// TIA Portal V17 export
// export: Created 2023-12-22T15:08:00.0545629Z, ExportSetting WithDefaults, DisplayName Totally Integrated Automation Portal, DisplayVersion V17, DisplayName TIA Portal Openness, DisplayVersion V17, DisplayName TIA Portal Version Control Interface, DisplayVersion V17, DisplayName STEP 7 Professional, DisplayVersion V17, DisplayName STEP 7 Safety, DisplayVersion V17, DisplayName WinCC Advanced, DisplayVersion V17
FUNCTION_BLOCK "PS_One"   // FB11, LAD
{ S7_Optimized_Access := 'FALSE' }
VERSION : 0.1
// Mode - 0 - выкл, 1 - быстрый разгон, 2 - плавный разон, 3 - работа, 4 - притормозить для ввода нового насоса, 5 - замедлить плавно, 6 - замедлить быстро
// 
// Status - 0 выкл, 1 - быстро разгоняется, 10 - вышел на точку, 2 - плавно разгоняется, 20 - вышел на точку, 3 - в работе, 4 - притормаживается для выхода на общую точку, 40 - общая точка достигнута, 5 - замедлить для отключения, 50 - замедлено до нижней точки, 6 - вывести из работы через быстрый сброс оборотов, 60 - обороты сброшены и готов к отключению, 99 - насос в аварии/не готов к работе
// stored: AutoNumber false, IsIECCheckEnabled false, SetENOAutomatically false, UDAEnableTagReadback false
   VAR_INPUT
      in_PE : Real;   // Давление на всасывании
      P_FB_SP : Real;   // Текущая скорость / Уставка скорости для ЧП
      P_Alarm : Bool;   // Авария ЧП
      P_Warning : Bool;   // Предупреждение ЧП
   END_VAR
   VAR_OUTPUT
      P_CMD : Bool;   // Команда на ЧП
      P_SP : Real;   // Уставка на ЧП
      P_Step_Up : Real := 0.01;   // Шаг разгона для ЧП
      P_Step_Down : Real := 0.01;   // Шаг замедления для ЧП
   END_VAR
   VAR_IN_OUT
      P_Res : DInt;   // Наработка ЧП
   END_VAR
   VAR DB_SPECIFIC
      CMD : "CMD";   // Блок команд
      Min { S7_SetPoint := 'True'} : Bool;
      Max : Bool;
      PE_Warning : Bool;
      SP_A : Real;   // Уставка в авторежиме
      SP : Real;   // Фактическая уставка
      Mode : Int;   // Запрашиваемый режим работы
      Hand_Mode : Int := 3;   // Режим работы в ручном режиме
      Status : Int;   // Фактический режим работы
      Weight : Real;   // Коэфф. выбора насоса
      Start_per_H_SP : Int := 5;
      Start_per_H_Now : Int;
      Alarms : Word;
      Events : Word;
      pos : Array[0..15] of Bool;
   END_VAR
   VAR
      T_Delay { S7_SetPoint := 'True'} : "Time_M";   // Минимальная задержка между пусками
      T_PE_Delay { S7_SetPoint := 'True'} : "Time_M";
   END_VAR
   VAR_TEMP
      ev : Bool;
   END_VAR
   // T_Delay.SP_M := 10;
   // T_Delay.SP_S := 0;
   VAR_TEMP   // added for the SCL form of the ladder/FBD networks
      _w1 : Bool;
      _w2 : Bool;
      _w3 : Bool;
      _w4 : Bool;
      _w5 : Bool;
      _w6 : Bool;
      _w7 : Bool;
      _w8 : Bool;
      _w9 : Bool;
      _w10 : Bool;
      _w11 : Bool;
      _w12 : Bool;
      _w13 : Bool;
      _w14 : Bool;
      _w15 : Bool;
      _w16 : Bool;
      _w17 : Bool;
      _w18 : Bool;
      _w19 : Bool;
      _w20 : Bool;
   END_VAR
BEGIN

REGION Network 1: - - -
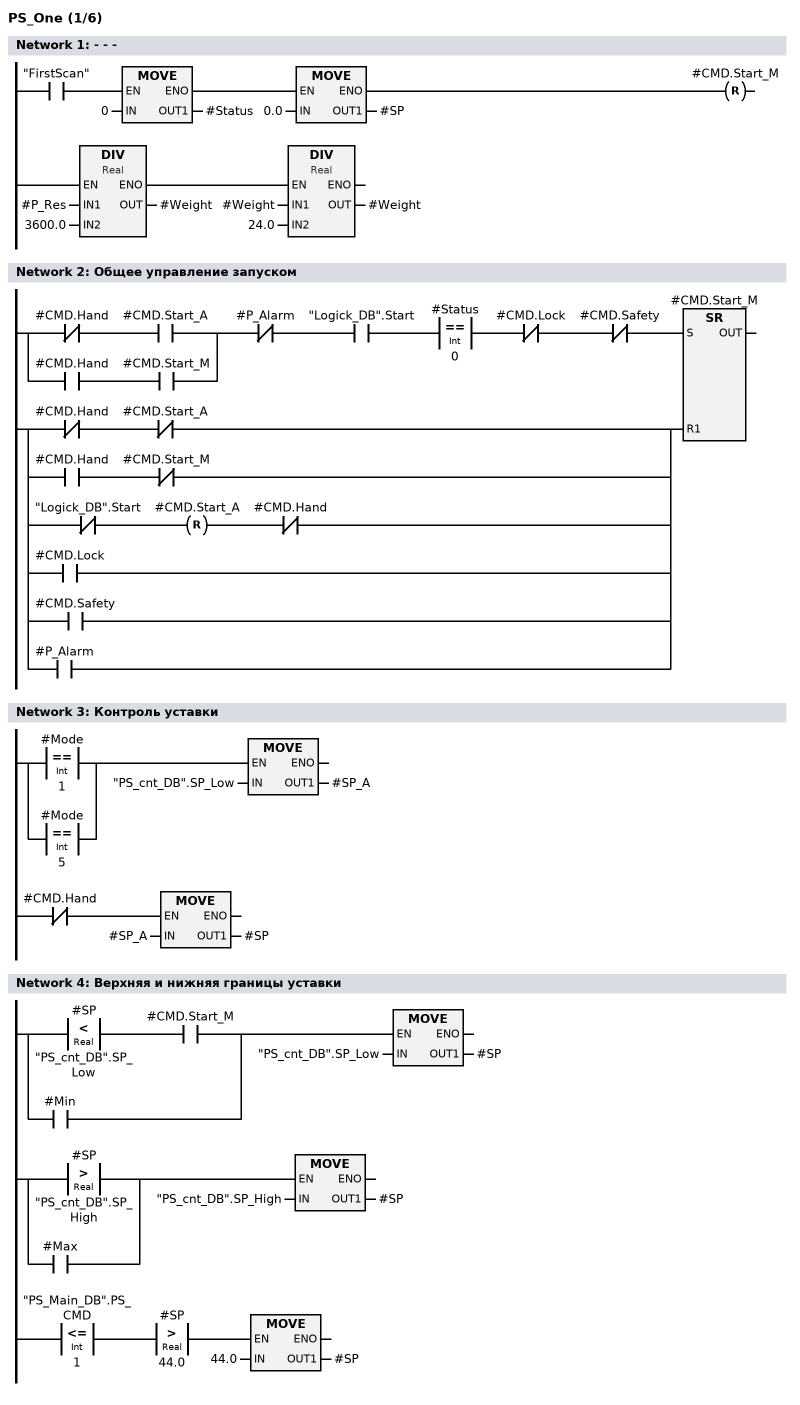
   RUNG wire#powerrail
      Contact( "FirstScan" )
      Move(in := 0, out1 => #Status)
      Move(in := 0.0, out1 => #SP)
      R_Coil( #CMD.Start_M )
   END_RUNG
   RUNG wire#powerrail
      { S7_Templates := "SrcType := Real" } Div(in1 := #P_Res, in2 := 3600.0, out => #Weight)
      { S7_Templates := "SrcType := Real" } Div(in1 := #Weight, in2 := 24.0, out => #Weight)
   END_RUNG
   // the same network as SCL:
   IF "FirstScan" THEN
       #Status := 0;
       #SP := 0.0;
       #CMD.Start_M := FALSE;
   END_IF;
   #Weight := #P_Res / 3600.0;
   #Weight := #Weight / 24.0;
END_REGION

REGION Network 2: Общее управление запуском
   RUNG wire#powerrail
      I_Contact( #CMD.Hand )
      Contact( #CMD.Start_A )
      wire#w1
      I_Contact( #P_Alarm )
      Contact( "Logick_DB".Start )
      { S7_Templates := "SrcType := Int" } EQ_Contact(in1 := #Status, in2 := 0)
      I_Contact( #CMD.Lock )
      I_Contact( #CMD.Safety )
      S_SR(operand := #CMD.Start_M, r1 := wire#w2)
   END_RUNG
   RUNG wire#powerrail
      Contact( #CMD.Hand )
      Contact( #CMD.Start_M )
   END_RUNG wire#w1
   RUNG wire#powerrail
      I_Contact( #CMD.Hand )
      I_Contact( #CMD.Start_A )
   END_RUNG wire#w2
   RUNG wire#powerrail
      Contact( #CMD.Hand )
      I_Contact( #CMD.Start_M )
   END_RUNG wire#w2
   RUNG wire#powerrail
      I_Contact( "Logick_DB".Start )
      R_Coil( #CMD.Start_A )
      I_Contact( #CMD.Hand )
   END_RUNG wire#w2
   RUNG wire#powerrail
      Contact( #CMD.Lock )
   END_RUNG wire#w2
   RUNG wire#powerrail
      Contact( #CMD.Safety )
   END_RUNG wire#w2
   RUNG wire#powerrail
      Contact( #P_Alarm )
   END_RUNG wire#w2
   // the same network as SCL:
   #_w1 := ((NOT #CMD.Hand AND #CMD.Start_A) OR (#CMD.Hand AND #CMD.Start_M)) AND NOT #P_Alarm AND "Logick_DB".Start AND (#Status = 0) AND NOT #CMD.Lock AND NOT #CMD.Safety;
   #_w2 := NOT #CMD.Hand AND NOT #CMD.Start_A;
   IF NOT "Logick_DB".Start THEN #CMD.Start_A := FALSE; END_IF;
   #_w3 := #_w2 OR (#CMD.Hand AND NOT #CMD.Start_M) OR (NOT "Logick_DB".Start AND NOT #CMD.Hand) OR #CMD.Lock OR #CMD.Safety OR #P_Alarm;
   IF #_w1 THEN
       #CMD.Start_M := TRUE;   // SR flip-flop
   END_IF;
   IF #_w3 THEN #CMD.Start_M := FALSE; END_IF;
END_REGION

REGION Network 3: Контроль уставки
   RUNG wire#powerrail
      { S7_Templates := "SrcType := Int" } EQ_Contact(in1 := #Mode, in2 := 1)
      wire#w1
      Move(in := "PS_cnt_DB".SP_Low, out1 => #SP_A)
   END_RUNG
   RUNG wire#powerrail
      { S7_Templates := "SrcType := Int" } EQ_Contact(in1 := #Mode, in2 := 5)
   END_RUNG wire#w1
   RUNG wire#powerrail
      I_Contact( #CMD.Hand )
      Move(in := #SP_A, out1 => #SP)
   END_RUNG
   // the same network as SCL:
   IF (#Mode = 1) OR (#Mode = 5) THEN #SP_A := "PS_cnt_DB".SP_Low; END_IF;
   IF NOT #CMD.Hand THEN #SP := #SP_A; END_IF;
END_REGION

REGION Network 4: Верхняя и нижняя границы уставки
   RUNG wire#powerrail
      { S7_Templates := "SrcType := Real" } LT_Contact(in1 := #SP, in2 := "PS_cnt_DB".SP_Low)
      Contact( #CMD.Start_M )
      wire#w1
      Move(in := "PS_cnt_DB".SP_Low, out1 => #SP)
   END_RUNG
   RUNG wire#powerrail
      Contact( #Min )
   END_RUNG wire#w1
   RUNG wire#powerrail
      { S7_Templates := "SrcType := Real" } GT_Contact(in1 := #SP, in2 := "PS_cnt_DB".SP_High)
      wire#w2
      Move(in := "PS_cnt_DB".SP_High, out1 => #SP)
   END_RUNG
   RUNG wire#powerrail
      Contact( #Max )
   END_RUNG wire#w2
   RUNG wire#powerrail
      { S7_Templates := "SrcType := Int" } LE_Contact(in1 := "PS_Main_DB".PS_CMD, in2 := 1)
      { S7_Templates := "SrcType := Real" } GT_Contact(in1 := #SP, in2 := 44.0)
      Move(in := 44.0, out1 => #SP)
   END_RUNG
   // the same network as SCL:
   IF ((#SP < "PS_cnt_DB".SP_Low) AND #CMD.Start_M) OR #Min THEN #SP := "PS_cnt_DB".SP_Low; END_IF;
   IF (#SP > "PS_cnt_DB".SP_High) OR #Max THEN #SP := "PS_cnt_DB".SP_High; END_IF;
   IF ("PS_Main_DB".PS_CMD <= 1) AND (#SP > 44.0) THEN #SP := 44.0; END_IF;
END_REGION

REGION Network 5
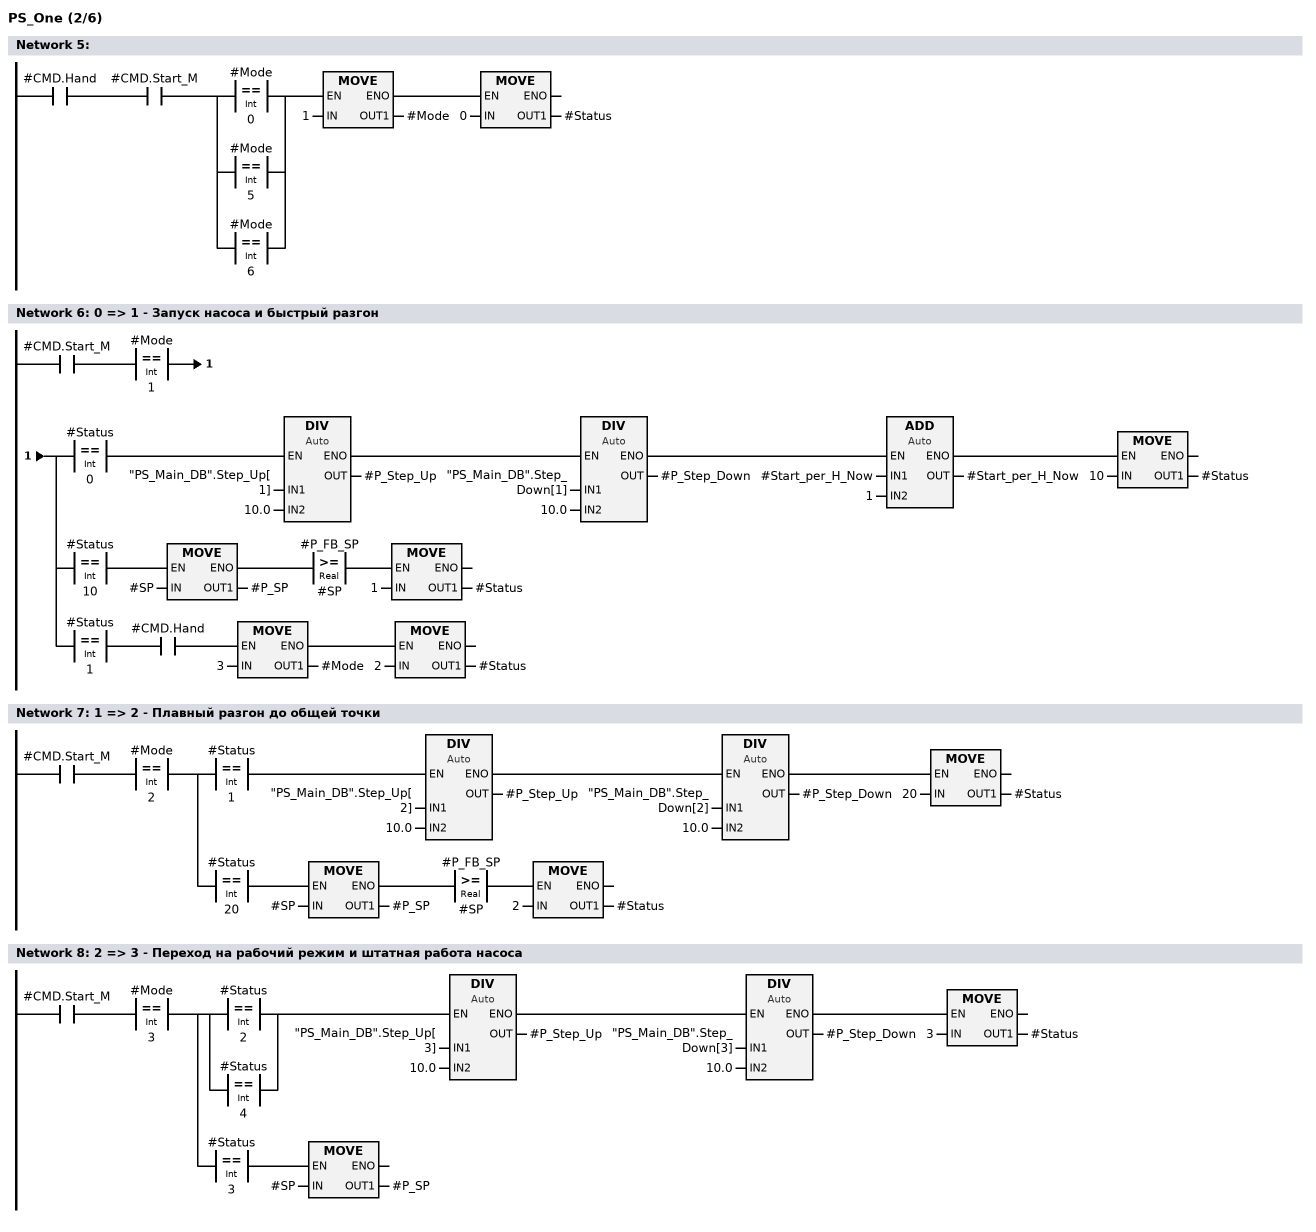
   RUNG wire#powerrail
      Contact( #CMD.Hand )
      Contact( #CMD.Start_M )
      wire#w1
      { S7_Templates := "SrcType := Int" } EQ_Contact(in1 := #Mode, in2 := 0)
      wire#w2
      Move(in := 1, out1 => #Mode)
      Move(in := 0, out1 => #Status)
   END_RUNG
   RUNG wire#w1
      { S7_Templates := "SrcType := Int" } EQ_Contact(in1 := #Mode, in2 := 5)
   END_RUNG wire#w2
   RUNG wire#w1
      { S7_Templates := "SrcType := Int" } EQ_Contact(in1 := #Mode, in2 := 6)
   END_RUNG wire#w2
   // the same network as SCL:
   #_w1 := #CMD.Hand AND #CMD.Start_M AND ((#Mode = 0) OR (#Mode = 5) OR (#Mode = 6));
   IF #_w1 THEN
       #Mode := 1;
       #Status := 0;
   END_IF;
END_REGION

REGION Network 6: 0 => 1 - Запуск насоса и быстрый разгон
   RUNG wire#powerrail
      Contact( #CMD.Start_M )
      { S7_Templates := "SrcType := Int" } EQ_Contact(in1 := #Mode, in2 := 1)
      wire#w1
      { S7_Templates := "SrcType := Int" } EQ_Contact(in1 := #Status, in2 := 0)
      Div(in1 := "PS_Main_DB".Step_Up[1], in2 := 10.0, out => #P_Step_Up)
      Div(in1 := "PS_Main_DB".Step_Down[1], in2 := 10.0, out => #P_Step_Down)
      Add(in1 := #Start_per_H_Now, in2 := 1, out => #Start_per_H_Now)
      Move(in := 10, out1 => #Status)
   END_RUNG
   RUNG wire#w1
      { S7_Templates := "SrcType := Int" } EQ_Contact(in1 := #Status, in2 := 10)
      Move(in := #SP, out1 => #P_SP)
      { S7_Templates := "SrcType := Real" } GE_Contact(in1 := #P_FB_SP, in2 := #SP)
      Move(in := 1, out1 => #Status)
   END_RUNG
   RUNG wire#w1
      { S7_Templates := "SrcType := Int" } EQ_Contact(in1 := #Status, in2 := 1)
      Contact( #CMD.Hand )
      Move(in := 3, out1 => #Mode)
      Move(in := 2, out1 => #Status)
   END_RUNG
   // the same network as SCL:
   #_w1 := #CMD.Start_M AND (#Mode = 1);
   IF #_w1 AND (#Status = 0) THEN
       #P_Step_Up := "PS_Main_DB".Step_Up[1] / 10.0;
       #P_Step_Down := "PS_Main_DB".Step_Down[1] / 10.0;
       #Start_per_H_Now := #Start_per_H_Now + 1;
       #Status := 10;
   END_IF;
   #_w2 := #_w1 AND (#Status = 10);
   IF #_w2 THEN #P_SP := #SP; END_IF;
   IF #_w2 AND (#P_FB_SP >= #SP) THEN #Status := 1; END_IF;
   IF #_w1 AND (#Status = 1) AND #CMD.Hand THEN
       #Mode := 3;
       #Status := 2;
   END_IF;
END_REGION

REGION Network 7: 1 => 2 - Плавный разгон до общей точки
   RUNG wire#powerrail
      Contact( #CMD.Start_M )
      { S7_Templates := "SrcType := Int" } EQ_Contact(in1 := #Mode, in2 := 2)
      wire#w1
      { S7_Templates := "SrcType := Int" } EQ_Contact(in1 := #Status, in2 := 1)
      Div(in1 := "PS_Main_DB".Step_Up[2], in2 := 10.0, out => #P_Step_Up)
      Div(in1 := "PS_Main_DB".Step_Down[2], in2 := 10.0, out => #P_Step_Down)
      Move(in := 20, out1 => #Status)
   END_RUNG
   RUNG wire#w1
      { S7_Templates := "SrcType := Int" } EQ_Contact(in1 := #Status, in2 := 20)
      Move(in := #SP, out1 => #P_SP)
      { S7_Templates := "SrcType := Real" } GE_Contact(in1 := #P_FB_SP, in2 := #SP)
      Move(in := 2, out1 => #Status)
   END_RUNG
   // the same network as SCL:
   #_w1 := #CMD.Start_M AND (#Mode = 2);
   IF #_w1 AND (#Status = 1) THEN
       #P_Step_Up := "PS_Main_DB".Step_Up[2] / 10.0;
       #P_Step_Down := "PS_Main_DB".Step_Down[2] / 10.0;
       #Status := 20;
   END_IF;
   #_w2 := #_w1 AND (#Status = 20);
   IF #_w2 THEN #P_SP := #SP; END_IF;
   IF #_w2 AND (#P_FB_SP >= #SP) THEN #Status := 2; END_IF;
END_REGION

REGION Network 8: 2 => 3 - Переход на рабочий режим и штатная работа насоса
   RUNG wire#powerrail
      Contact( #CMD.Start_M )
      { S7_Templates := "SrcType := Int" } EQ_Contact(in1 := #Mode, in2 := 3)
      wire#w1
      { S7_Templates := "SrcType := Int" } EQ_Contact(in1 := #Status, in2 := 2)
      wire#w2
      Div(in1 := "PS_Main_DB".Step_Up[3], in2 := 10.0, out => #P_Step_Up)
      Div(in1 := "PS_Main_DB".Step_Down[3], in2 := 10.0, out => #P_Step_Down)
      Move(in := 3, out1 => #Status)
   END_RUNG
   RUNG wire#w1
      { S7_Templates := "SrcType := Int" } EQ_Contact(in1 := #Status, in2 := 4)
   END_RUNG wire#w2
   RUNG wire#w1
      { S7_Templates := "SrcType := Int" } EQ_Contact(in1 := #Status, in2 := 3)
      Move(in := #SP, out1 => #P_SP)
   END_RUNG
   // the same network as SCL:
   #_w1 := #CMD.Start_M AND (#Mode = 3);
   IF #_w1 AND ((#Status = 2) OR (#Status = 4)) THEN
       #P_Step_Up := "PS_Main_DB".Step_Up[3] / 10.0;
       #P_Step_Down := "PS_Main_DB".Step_Down[3] / 10.0;
       #Status := 3;
   END_IF;
   IF #_w1 AND (#Status = 3) THEN #P_SP := #SP; END_IF;
END_REGION

REGION Network 9: 3 => 4 - Снижение скорости для подключения нового насоса
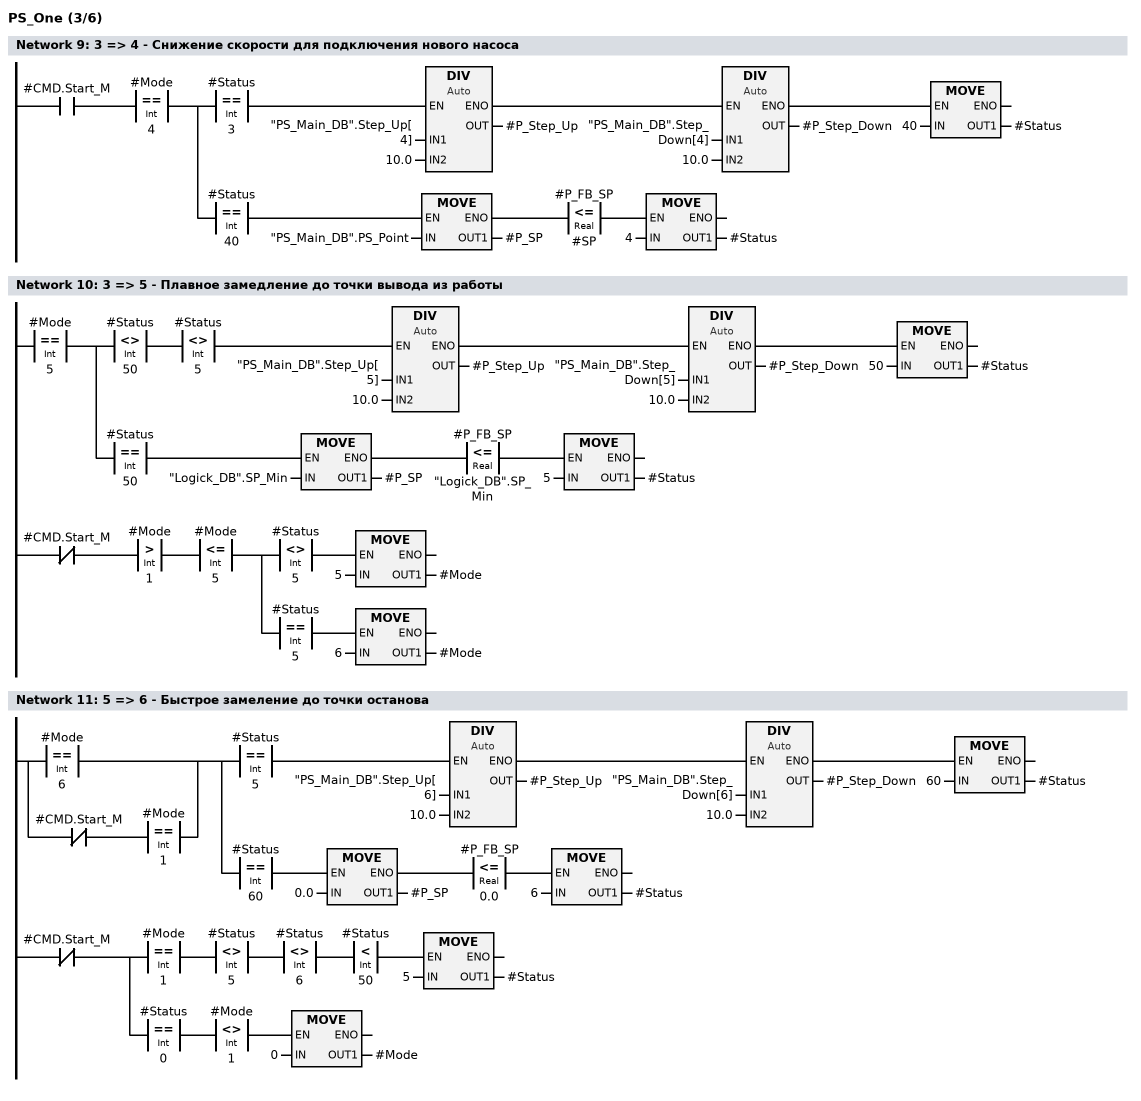
   RUNG wire#powerrail
      Contact( #CMD.Start_M )
      { S7_Templates := "SrcType := Int" } EQ_Contact(in1 := #Mode, in2 := 4)
      wire#w1
      { S7_Templates := "SrcType := Int" } EQ_Contact(in1 := #Status, in2 := 3)
      Div(in1 := "PS_Main_DB".Step_Up[4], in2 := 10.0, out => #P_Step_Up)
      Div(in1 := "PS_Main_DB".Step_Down[4], in2 := 10.0, out => #P_Step_Down)
      Move(in := 40, out1 => #Status)
   END_RUNG
   RUNG wire#w1
      { S7_Templates := "SrcType := Int" } EQ_Contact(in1 := #Status, in2 := 40)
      Move(in := "PS_Main_DB".PS_Point, out1 => #P_SP)
      { S7_Templates := "SrcType := Real" } LE_Contact(in1 := #P_FB_SP, in2 := #SP)
      Move(in := 4, out1 => #Status)
   END_RUNG
   // the same network as SCL:
   #_w1 := #CMD.Start_M AND (#Mode = 4);
   IF #_w1 AND (#Status = 3) THEN
       #P_Step_Up := "PS_Main_DB".Step_Up[4] / 10.0;
       #P_Step_Down := "PS_Main_DB".Step_Down[4] / 10.0;
       #Status := 40;
   END_IF;
   #_w2 := #_w1 AND (#Status = 40);
   IF #_w2 THEN #P_SP := "PS_Main_DB".PS_Point; END_IF;
   IF #_w2 AND (#P_FB_SP <= #SP) THEN #Status := 4; END_IF;
END_REGION

REGION Network 10: 3 => 5 - Плавное замедление до точки вывода из работы
   RUNG wire#powerrail
      { S7_Templates := "SrcType := Int" } EQ_Contact(in1 := #Mode, in2 := 5)
      wire#w1
      { S7_Templates := "SrcType := Int" } NE_Contact(in1 := #Status, in2 := 50)
      { S7_Templates := "SrcType := Int" } NE_Contact(in1 := #Status, in2 := 5)
      Div(in1 := "PS_Main_DB".Step_Up[5], in2 := 10.0, out => #P_Step_Up)
      Div(in1 := "PS_Main_DB".Step_Down[5], in2 := 10.0, out => #P_Step_Down)
      Move(in := 50, out1 => #Status)
   END_RUNG
   RUNG wire#w1
      { S7_Templates := "SrcType := Int" } EQ_Contact(in1 := #Status, in2 := 50)
      Move(in := "Logick_DB".SP_Min, out1 => #P_SP)
      { S7_Templates := "SrcType := Real" } LE_Contact(in1 := #P_FB_SP, in2 := "Logick_DB".SP_Min)
      Move(in := 5, out1 => #Status)
   END_RUNG
   RUNG wire#powerrail
      I_Contact( #CMD.Start_M )
      { S7_Templates := "SrcType := Int" } GT_Contact(in1 := #Mode, in2 := 1)
      { S7_Templates := "SrcType := Int" } LE_Contact(in1 := #Mode, in2 := 5)
      wire#w2
      { S7_Templates := "SrcType := Int" } NE_Contact(in1 := #Status, in2 := 5)
      Move(in := 5, out1 => #Mode)
   END_RUNG
   RUNG wire#w2
      { S7_Templates := "SrcType := Int" } EQ_Contact(in1 := #Status, in2 := 5)
      Move(in := 6, out1 => #Mode)
   END_RUNG
   // the same network as SCL:
   #_w1 := #Mode = 5;
   IF #_w1 AND (#Status <> 50) AND (#Status <> 5) THEN
       #P_Step_Up := "PS_Main_DB".Step_Up[5] / 10.0;
       #P_Step_Down := "PS_Main_DB".Step_Down[5] / 10.0;
       #Status := 50;
   END_IF;
   #_w2 := #_w1 AND (#Status = 50);
   IF #_w2 THEN #P_SP := "Logick_DB".SP_Min; END_IF;
   IF #_w2 AND (#P_FB_SP <= "Logick_DB".SP_Min) THEN #Status := 5; END_IF;
   #_w3 := NOT #CMD.Start_M AND (#Mode > 1) AND (#Mode <= 5);
   IF #_w3 AND (#Status <> 5) THEN #Mode := 5; END_IF;
   IF #_w3 AND (#Status = 5) THEN #Mode := 6; END_IF;
END_REGION

REGION Network 11: 5 => 6 - Быстрое замеление до точки останова
   RUNG wire#powerrail
      { S7_Templates := "SrcType := Int" } EQ_Contact(in1 := #Mode, in2 := 6)
      wire#w1
      { S7_Templates := "SrcType := Int" } EQ_Contact(in1 := #Status, in2 := 5)
      Div(in1 := "PS_Main_DB".Step_Up[6], in2 := 10.0, out => #P_Step_Up)
      Div(in1 := "PS_Main_DB".Step_Down[6], in2 := 10.0, out => #P_Step_Down)
      Move(in := 60, out1 => #Status)
   END_RUNG
   RUNG wire#powerrail
      I_Contact( #CMD.Start_M )
      { S7_Templates := "SrcType := Int" } EQ_Contact(in1 := #Mode, in2 := 1)
   END_RUNG wire#w1
   RUNG wire#w1
      { S7_Templates := "SrcType := Int" } EQ_Contact(in1 := #Status, in2 := 60)
      Move(in := 0.0, out1 => #P_SP)
      { S7_Templates := "SrcType := Real" } LE_Contact(in1 := #P_FB_SP, in2 := 0.0)
      Move(in := 6, out1 => #Status)
   END_RUNG
   RUNG wire#powerrail
      I_Contact( #CMD.Start_M )
      wire#w2
      { S7_Templates := "SrcType := Int" } EQ_Contact(in1 := #Mode, in2 := 1)
      { S7_Templates := "SrcType := Int" } NE_Contact(in1 := #Status, in2 := 5)
      { S7_Templates := "SrcType := Int" } NE_Contact(in1 := #Status, in2 := 6)
      { S7_Templates := "SrcType := Int" } LT_Contact(in1 := #Status, in2 := 50)
      Move(in := 5, out1 => #Status)
   END_RUNG
   RUNG wire#w2
      { S7_Templates := "SrcType := Int" } EQ_Contact(in1 := #Status, in2 := 0)
      { S7_Templates := "SrcType := Int" } NE_Contact(in1 := #Mode, in2 := 1)
      Move(in := 0, out1 => #Mode)
   END_RUNG
   // the same network as SCL:
   #_w1 := (#Mode = 6) OR (NOT #CMD.Start_M AND (#Mode = 1));
   IF #_w1 AND (#Status = 5) THEN
       #P_Step_Up := "PS_Main_DB".Step_Up[6] / 10.0;
       #P_Step_Down := "PS_Main_DB".Step_Down[6] / 10.0;
       #Status := 60;
   END_IF;
   #_w2 := #_w1 AND (#Status = 60);
   IF #_w2 THEN #P_SP := 0.0; END_IF;
   IF #_w2 AND (#P_FB_SP <= 0.0) THEN #Status := 6; END_IF;
   IF NOT #CMD.Start_M AND (#Mode = 1) AND (#Status <> 5) AND (#Status <> 6) AND (#Status < 50) THEN
       #Status := 5;
   END_IF;
   IF NOT #CMD.Start_M AND (#Status = 0) AND (#Mode <> 1) THEN #Mode := 0; END_IF;
END_REGION

REGION Network 12: 6 => 0 - Насос успешно остановлен
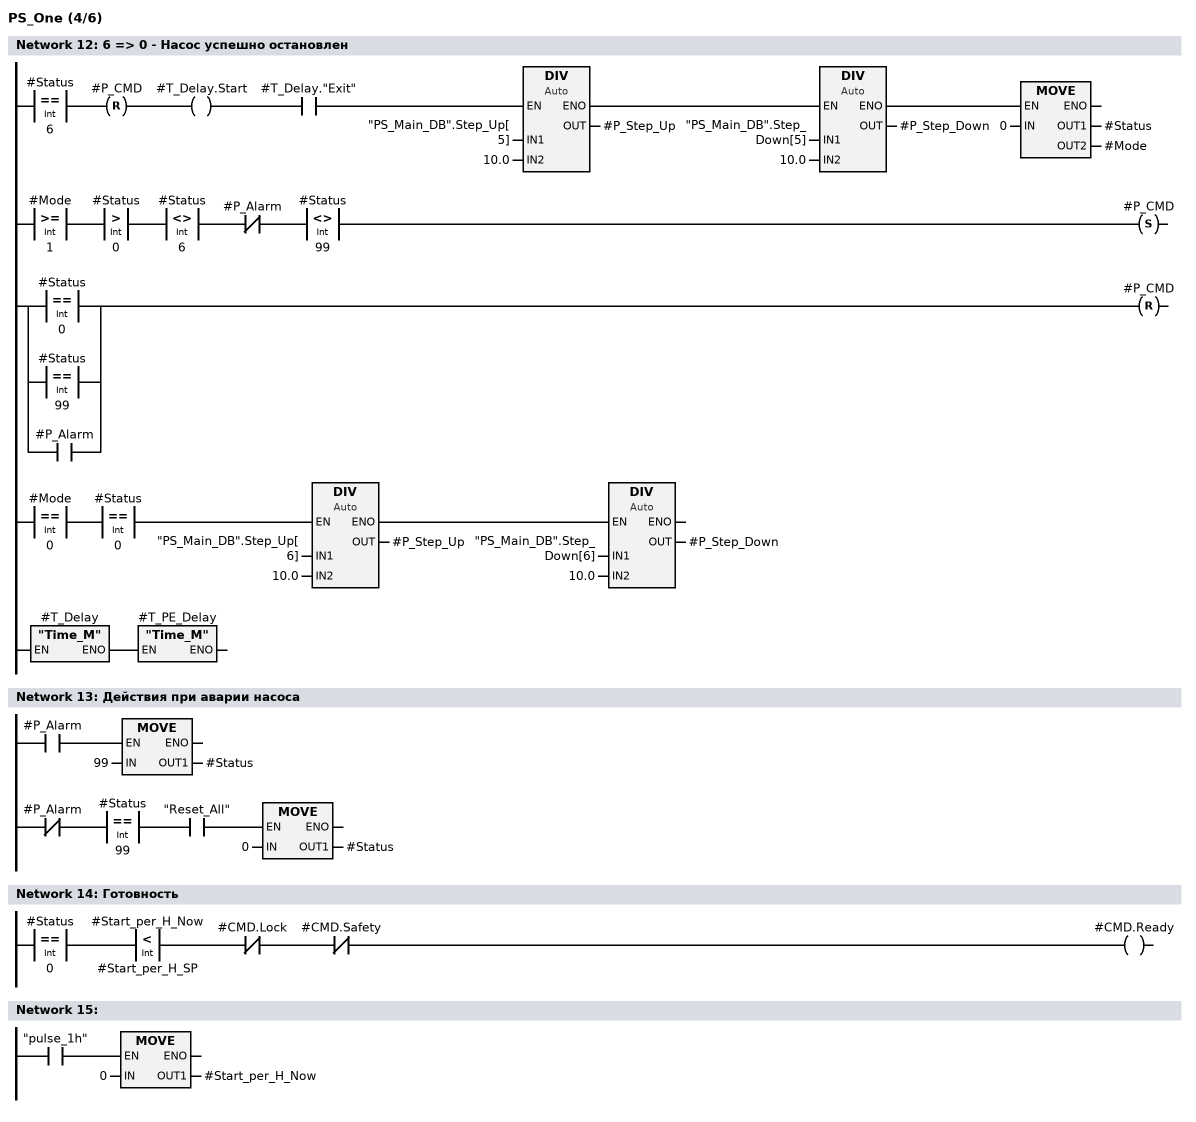
   RUNG wire#powerrail
      { S7_Templates := "SrcType := Int" } EQ_Contact(in1 := #Status, in2 := 6)
      R_Coil( #P_CMD )
      Coil( #T_Delay.Start )
      Contact( #T_Delay."Exit" )
      Div(in1 := "PS_Main_DB".Step_Up[5], in2 := 10.0, out => #P_Step_Up)
      Div(in1 := "PS_Main_DB".Step_Down[5], in2 := 10.0, out => #P_Step_Down)
      Move(in := 0, out1 => #Status, out2 => #Mode)
   END_RUNG
   RUNG wire#powerrail
      { S7_Templates := "SrcType := Int" } GE_Contact(in1 := #Mode, in2 := 1)
      { S7_Templates := "SrcType := Int" } GT_Contact(in1 := #Status, in2 := 0)
      { S7_Templates := "SrcType := Int" } NE_Contact(in1 := #Status, in2 := 6)
      I_Contact( #P_Alarm )
      { S7_Templates := "SrcType := Int" } NE_Contact(in1 := #Status, in2 := 99)
      S_Coil( #P_CMD )
   END_RUNG
   RUNG wire#powerrail
      { S7_Templates := "SrcType := Int" } EQ_Contact(in1 := #Status, in2 := 0)
      wire#w1
      R_Coil( #P_CMD )
   END_RUNG
   RUNG wire#powerrail
      { S7_Templates := "SrcType := Int" } EQ_Contact(in1 := #Status, in2 := 99)
   END_RUNG wire#w1
   RUNG wire#powerrail
      Contact( #P_Alarm )
   END_RUNG wire#w1
   RUNG wire#powerrail
      { S7_Templates := "SrcType := Int" } EQ_Contact(in1 := #Mode, in2 := 0)
      { S7_Templates := "SrcType := Int" } EQ_Contact(in1 := #Status, in2 := 0)
      Div(in1 := "PS_Main_DB".Step_Up[6], in2 := 10.0, out => #P_Step_Up)
      Div(in1 := "PS_Main_DB".Step_Down[6], in2 := 10.0, out => #P_Step_Down)
   END_RUNG
   RUNG wire#powerrail
      #T_Delay()
      #T_PE_Delay()
   END_RUNG
   // the same network as SCL:
   #_w1 := #Status = 6;
   IF #_w1 THEN #P_CMD := FALSE; END_IF;
   #T_Delay.Start := #_w1;
   IF #_w1 AND #T_Delay."Exit" THEN
       #P_Step_Up := "PS_Main_DB".Step_Up[5] / 10.0;
       #P_Step_Down := "PS_Main_DB".Step_Down[5] / 10.0;
       #Status := 0;
       #Mode := 0;
   END_IF;
   IF (#Mode >= 1) AND (#Status > 0) AND (#Status <> 6) AND NOT #P_Alarm AND (#Status <> 99) THEN
       #P_CMD := TRUE;
   END_IF;
   IF (#Status = 0) OR (#Status = 99) OR #P_Alarm THEN #P_CMD := FALSE; END_IF;
   IF (#Mode = 0) AND (#Status = 0) THEN
       #P_Step_Up := "PS_Main_DB".Step_Up[6] / 10.0;
       #P_Step_Down := "PS_Main_DB".Step_Down[6] / 10.0;
   END_IF;
   #T_Delay(ENO => #_w2);   // "Time_M"
   IF #_w2 THEN
       #T_PE_Delay();   // "Time_M"
   END_IF;
END_REGION

REGION Network 13: Действия при аварии насоса
   RUNG wire#powerrail
      Contact( #P_Alarm )
      Move(in := 99, out1 => #Status)
   END_RUNG
   RUNG wire#powerrail
      I_Contact( #P_Alarm )
      { S7_Templates := "SrcType := Int" } EQ_Contact(in1 := #Status, in2 := 99)
      Contact( "Reset_All" )
      Move(in := 0, out1 => #Status)
   END_RUNG
   // the same network as SCL:
   IF #P_Alarm THEN #Status := 99; END_IF;
   IF NOT #P_Alarm AND (#Status = 99) AND "Reset_All" THEN #Status := 0; END_IF;
END_REGION

REGION Network 14: Готовность
   RUNG wire#powerrail
      { S7_Templates := "SrcType := Int" } EQ_Contact(in1 := #Status, in2 := 0)
      { S7_Templates := "SrcType := Int" } LT_Contact(in1 := #Start_per_H_Now, in2 := #Start_per_H_SP)
      I_Contact( #CMD.Lock )
      I_Contact( #CMD.Safety )
      Coil( #CMD.Ready )
   END_RUNG
   // the same network as SCL:
   #CMD.Ready := (#Status = 0) AND (#Start_per_H_Now < #Start_per_H_SP) AND NOT #CMD.Lock AND NOT #CMD.Safety;
END_REGION

REGION Network 15
   RUNG wire#powerrail
      Contact( "pulse_1h" )
      Move(in := 0, out1 => #Start_per_H_Now)
   END_RUNG
   // the same network as SCL:
   IF "pulse_1h" THEN #Start_per_H_Now := 0; END_IF;
END_REGION

REGION Network 16
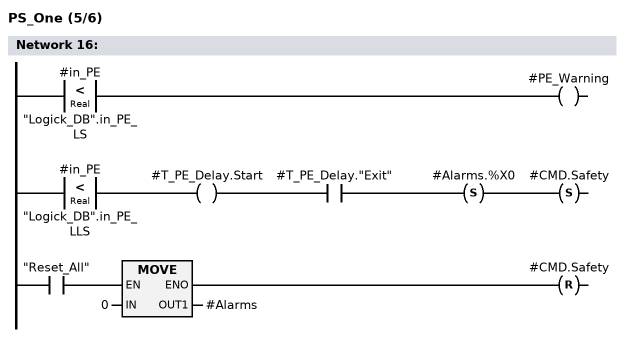
   RUNG wire#powerrail
      { S7_Templates := "SrcType := Real" } LT_Contact(in1 := #in_PE, in2 := "Logick_DB".in_PE_LS)
      Coil( #PE_Warning )
   END_RUNG
   RUNG wire#powerrail
      { S7_Templates := "SrcType := Real" } LT_Contact(in1 := #in_PE, in2 := "Logick_DB".in_PE_LLS)
      Coil( #T_PE_Delay.Start )
      Contact( #T_PE_Delay."Exit" )
      S_Coil( #Alarms.%X0 )
      S_Coil( #CMD.Safety )
   END_RUNG
   RUNG wire#powerrail
      Contact( "Reset_All" )
      Move(in := 0, out1 => #Alarms)
      R_Coil( #CMD.Safety )
   END_RUNG
   // the same network as SCL:
   #PE_Warning := #in_PE < "Logick_DB".in_PE_LS;
   #T_PE_Delay.Start := #in_PE < "Logick_DB".in_PE_LLS;
   IF #T_PE_Delay.Start AND #T_PE_Delay."Exit" THEN
       #Alarms.%X0 := TRUE;
       #CMD.Safety := TRUE;
   END_IF;
   IF "Reset_All" THEN
       #Alarms := 0;
       #CMD.Safety := FALSE;
   END_IF;
END_REGION

REGION Network 17: События привода
   // 0 - ручной режим активирован
   // 1 - ручной режим деактивирован
   // 2 - принудительный режим активирован
   // 3 - принудительный режим деактивирован
   // 4 - запуск в ручном режиме
   // 5 - останов в ручном режиме
   // 6 - местный режим управления активирован
   // 7 - местный режим управления деактивирован
   // 8 - запущено в местном режиме
   // 9 - остановлено в местном режиме
   // 10 - сервисный режим активирован
   // 11 - сервисный режим деактивирован
   // 12 - проведено сервисное обслуживание
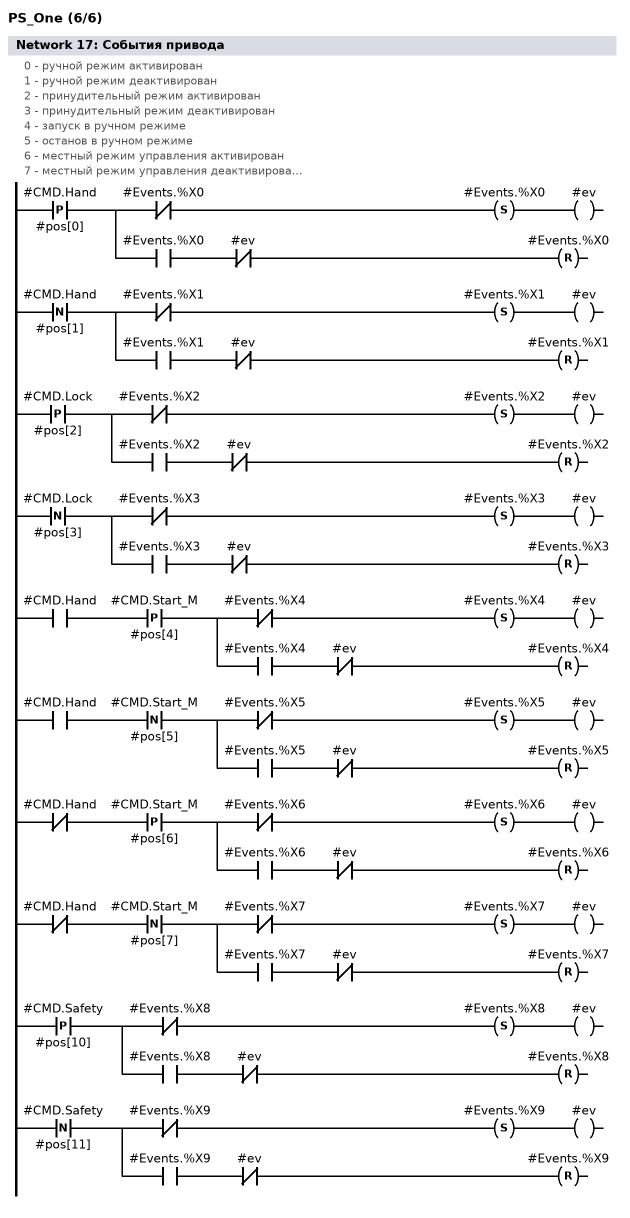
   RUNG wire#powerrail
      P_Contact(operand := #CMD.Hand, bit := #pos[0])
      wire#w1
      I_Contact( #Events.%X0 )
      S_Coil( #Events.%X0 )
      Coil( #ev )
   END_RUNG
   RUNG wire#w1
      Contact( #Events.%X0 )
      I_Contact( #ev )
      R_Coil( #Events.%X0 )
   END_RUNG
   RUNG wire#powerrail
      N_Contact(operand := #CMD.Hand, bit := #pos[1])
      wire#w2
      I_Contact( #Events.%X1 )
      S_Coil( #Events.%X1 )
      Coil( #ev )
   END_RUNG
   RUNG wire#w2
      Contact( #Events.%X1 )
      I_Contact( #ev )
      R_Coil( #Events.%X1 )
   END_RUNG
   RUNG wire#powerrail
      P_Contact(operand := #CMD.Lock, bit := #pos[2])
      wire#w3
      I_Contact( #Events.%X2 )
      S_Coil( #Events.%X2 )
      Coil( #ev )
   END_RUNG
   RUNG wire#w3
      Contact( #Events.%X2 )
      I_Contact( #ev )
      R_Coil( #Events.%X2 )
   END_RUNG
   RUNG wire#powerrail
      N_Contact(operand := #CMD.Lock, bit := #pos[3])
      wire#w4
      I_Contact( #Events.%X3 )
      S_Coil( #Events.%X3 )
      Coil( #ev )
   END_RUNG
   RUNG wire#w4
      Contact( #Events.%X3 )
      I_Contact( #ev )
      R_Coil( #Events.%X3 )
   END_RUNG
   RUNG wire#powerrail
      Contact( #CMD.Hand )
      P_Contact(operand := #CMD.Start_M, bit := #pos[4])
      wire#w5
      I_Contact( #Events.%X4 )
      S_Coil( #Events.%X4 )
      Coil( #ev )
   END_RUNG
   RUNG wire#w5
      Contact( #Events.%X4 )
      I_Contact( #ev )
      R_Coil( #Events.%X4 )
   END_RUNG
   RUNG wire#powerrail
      Contact( #CMD.Hand )
      N_Contact(operand := #CMD.Start_M, bit := #pos[5])
      wire#w6
      I_Contact( #Events.%X5 )
      S_Coil( #Events.%X5 )
      Coil( #ev )
   END_RUNG
   RUNG wire#w6
      Contact( #Events.%X5 )
      I_Contact( #ev )
      R_Coil( #Events.%X5 )
   END_RUNG
   RUNG wire#powerrail
      I_Contact( #CMD.Hand )
      P_Contact(operand := #CMD.Start_M, bit := #pos[6])
      wire#w7
      I_Contact( #Events.%X6 )
      S_Coil( #Events.%X6 )
      Coil( #ev )
   END_RUNG
   RUNG wire#w7
      Contact( #Events.%X6 )
      I_Contact( #ev )
      R_Coil( #Events.%X6 )
   END_RUNG
   RUNG wire#powerrail
      I_Contact( #CMD.Hand )
      N_Contact(operand := #CMD.Start_M, bit := #pos[7])
      wire#w8
      I_Contact( #Events.%X7 )
      S_Coil( #Events.%X7 )
      Coil( #ev )
   END_RUNG
   RUNG wire#w8
      Contact( #Events.%X7 )
      I_Contact( #ev )
      R_Coil( #Events.%X7 )
   END_RUNG
   RUNG wire#powerrail
      P_Contact(operand := #CMD.Safety, bit := #pos[10])
      wire#w9
      I_Contact( #Events.%X8 )
      S_Coil( #Events.%X8 )
      Coil( #ev )
   END_RUNG
   RUNG wire#w9
      Contact( #Events.%X8 )
      I_Contact( #ev )
      R_Coil( #Events.%X8 )
   END_RUNG
   RUNG wire#powerrail
      N_Contact(operand := #CMD.Safety, bit := #pos[11])
      wire#w10
      I_Contact( #Events.%X9 )
      S_Coil( #Events.%X9 )
      Coil( #ev )
   END_RUNG
   RUNG wire#w10
      Contact( #Events.%X9 )
      I_Contact( #ev )
      R_Coil( #Events.%X9 )
   END_RUNG
   // the same network as SCL:
   #_w1 := #CMD.Hand AND NOT #pos[0];   // rising edge of #CMD.Hand
   #pos[0] := #CMD.Hand;
   #_w2 := #_w1 AND NOT #Events.%X0;
   IF #_w2 THEN #Events.%X0 := TRUE; END_IF;
   #ev := #_w2;
   IF #_w1 AND #Events.%X0 AND NOT #ev THEN #Events.%X0 := FALSE; END_IF;
   #_w3 := NOT #CMD.Hand AND #pos[1];   // falling edge of #CMD.Hand
   #pos[1] := #CMD.Hand;
   #_w4 := #_w3 AND NOT #Events.%X1;
   IF #_w4 THEN #Events.%X1 := TRUE; END_IF;
   #ev := #_w4;
   IF #_w3 AND #Events.%X1 AND NOT #ev THEN #Events.%X1 := FALSE; END_IF;
   #_w5 := #CMD.Lock AND NOT #pos[2];   // rising edge of #CMD.Lock
   #pos[2] := #CMD.Lock;
   #_w6 := #_w5 AND NOT #Events.%X2;
   IF #_w6 THEN #Events.%X2 := TRUE; END_IF;
   #ev := #_w6;
   IF #_w5 AND #Events.%X2 AND NOT #ev THEN #Events.%X2 := FALSE; END_IF;
   #_w7 := NOT #CMD.Lock AND #pos[3];   // falling edge of #CMD.Lock
   #pos[3] := #CMD.Lock;
   #_w8 := #_w7 AND NOT #Events.%X3;
   IF #_w8 THEN #Events.%X3 := TRUE; END_IF;
   #ev := #_w8;
   IF #_w7 AND #Events.%X3 AND NOT #ev THEN #Events.%X3 := FALSE; END_IF;
   #_w9 := #CMD.Hand AND #CMD.Start_M AND NOT #pos[4];   // rising edge of #CMD.Start_M
   #pos[4] := #CMD.Start_M;
   #_w10 := #_w9 AND NOT #Events.%X4;
   IF #_w10 THEN #Events.%X4 := TRUE; END_IF;
   #ev := #_w10;
   IF #_w9 AND #Events.%X4 AND NOT #ev THEN #Events.%X4 := FALSE; END_IF;
   #_w11 := #CMD.Hand AND NOT #CMD.Start_M AND #pos[5];   // falling edge of #CMD.Start_M
   #pos[5] := #CMD.Start_M;
   #_w12 := #_w11 AND NOT #Events.%X5;
   IF #_w12 THEN #Events.%X5 := TRUE; END_IF;
   #ev := #_w12;
   IF #_w11 AND #Events.%X5 AND NOT #ev THEN #Events.%X5 := FALSE; END_IF;
   #_w13 := NOT #CMD.Hand AND #CMD.Start_M AND NOT #pos[6];   // rising edge of #CMD.Start_M
   #pos[6] := #CMD.Start_M;
   #_w14 := #_w13 AND NOT #Events.%X6;
   IF #_w14 THEN #Events.%X6 := TRUE; END_IF;
   #ev := #_w14;
   IF #_w13 AND #Events.%X6 AND NOT #ev THEN #Events.%X6 := FALSE; END_IF;
   #_w15 := NOT #CMD.Hand AND NOT #CMD.Start_M AND #pos[7];   // falling edge of #CMD.Start_M
   #pos[7] := #CMD.Start_M;
   #_w16 := #_w15 AND NOT #Events.%X7;
   IF #_w16 THEN #Events.%X7 := TRUE; END_IF;
   #ev := #_w16;
   IF #_w15 AND #Events.%X7 AND NOT #ev THEN #Events.%X7 := FALSE; END_IF;
   #_w17 := #CMD.Safety AND NOT #pos[10];   // rising edge of #CMD.Safety
   #pos[10] := #CMD.Safety;
   #_w18 := #_w17 AND NOT #Events.%X8;
   IF #_w18 THEN #Events.%X8 := TRUE; END_IF;
   #ev := #_w18;
   IF #_w17 AND #Events.%X8 AND NOT #ev THEN #Events.%X8 := FALSE; END_IF;
   #_w19 := NOT #CMD.Safety AND #pos[11];   // falling edge of #CMD.Safety
   #pos[11] := #CMD.Safety;
   #_w20 := #_w19 AND NOT #Events.%X9;
   IF #_w20 THEN #Events.%X9 := TRUE; END_IF;
   #ev := #_w20;
   IF #_w19 AND #Events.%X9 AND NOT #ev THEN #Events.%X9 := FALSE; END_IF;
END_REGION
END_FUNCTION_BLOCK
